// TIA Portal V17 export
// export: Created 2025-03-13T10:30:22.8196158Z, ExportSetting WithDefaults, DisplayName Totally Integrated Automation Portal, DisplayVersion V17 Update 8, DisplayName TIA Portal Openness, DisplayVersion V17 Update 8, DisplayName TIA Portal Version Control Interface, DisplayVersion V17, DisplayName SINAMICS Startdrive Advanced, DisplayVersion V17 SP2, DisplayName SINAMICS Startdrive G110M, G120, G120C, G120D, G120P, G115D, DisplayVersion V17 SP2, DisplayName SINAMICS Startdrive G130, G150, S120, S150, SINAMICS MV, S210, DisplayVersion V17 SP2, DisplayName STEP 7 Professional, DisplayVersion V17 Update 8, DisplayName SINUMERIK ONE STEP 7 Toolbox, DisplayVersion V17 Update 12, DisplayName SINUMERIK 840D sl STEP 7 Toolbox, DisplayVersion V17 Update 12, DisplayName STEP 7 Safety, DisplayVersion V17 Update 6, DisplayName WinCC Advanced, DisplayVersion V17 Update 8
FUNCTION "FC2390_ENERGY" : Void   // FC2390, LAD
{ S7_Optimized_Access := 'TRUE' }
VERSION : 0.1
// stored: AutoNumber false, IsIECCheckEnabled false, SetENOAutomatically false, UDAEnableTagReadback false
   VAR CONSTANT
      FC_NUMBER : DInt := 2390;
   END_VAR
BEGIN

REGION Network 1: CALL FC2391 SAVE ENERGY
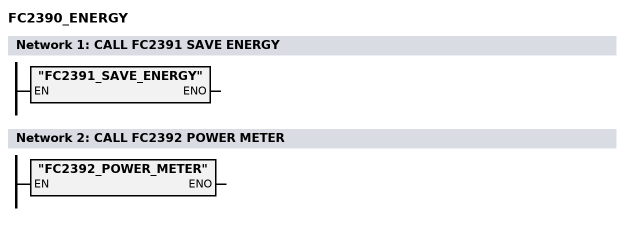
   RUNG wire#powerrail
      "FC2391_SAVE_ENERGY"()
   END_RUNG
   // the same network as SCL:
   "FC2391_SAVE_ENERGY"();
END_REGION

REGION Network 2: CALL FC2392 POWER METER
   RUNG wire#powerrail
      "FC2392_POWER_METER"()
   END_RUNG
   // the same network as SCL:
   "FC2392_POWER_METER"();
END_REGION
END_FUNCTION
